ABB RobotStudio station: PROYECTO_SIM_20221117-140459.rsstn

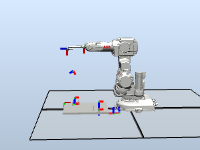
Station PROYECTO_SIM (saved by RobotStudio 6.5.7558.2005)
Controller IRB_140_6kg_0.81m
  mechanical unit ROB_1: IRB140_6_81_C_03, 6 joints, base frame (0, 0, 0) mm
Layout (positions relative to the parent item):
  - IRB140_6_81_C_03 [mechanism, from Robots\IRB140_6_81_C_G_03.rslib] at (0, 0, 0) mm; joint values [0, 0, 0, 0, 0, 0] (rad or m)
  - Herramienta_Proyecto [mechanism, from Libraries\Herramienta_Proyecto.rslib] at (515, 0, 712) mm, rotated rx 0 ry 90 rz 0 deg
  - Placa [part] at (500, 0, 0) mm
Attachment: Herramienta_Proyecto is attached to IRB140_6_81_C_03 / Link6
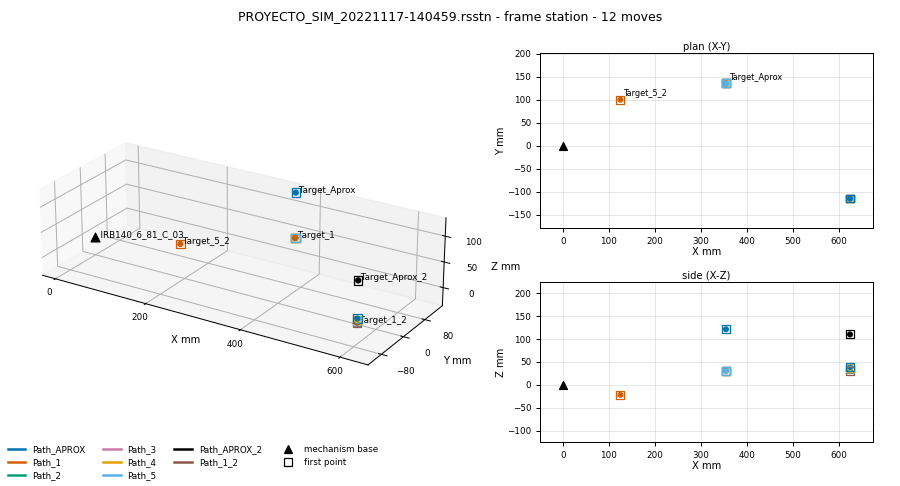
[picture p0: tool path of PROYECTO_SIM_20221117-140459.rsstn in frame station, 12 of 14 moves have a stored position in this frame; points joined in program order, loops and branches not executed]
Targets, tools, work objects and paths stored in the station, written as RAPID:
! task T_ROB1
MODULE CalibData
  PERS tooldata Herramienta_Proyecto_TCP:=[TRUE,[[20,0,187.132],[1,0,0,0]],[0.4,[8.3,90.3,0.6],[1,0,0,0],0,0,0]];
  TASK PERS wobjdata Workobject_1:=[FALSE,TRUE,"",[[750,-215,20],[0,0,1,0]],[[0,0,0],[1,0,0,0]]];
ENDMODULE

! task T_ROB1
MODULE Module1
  CONST jointtarget HOME:=[[0,0,0,0,0,0],[9E+09,9E+09,9E+09,9E+09,9E+09,9E+09]];
  CONST jointtarget MID:=[[0,30,0,0,0,0],[9E+09,9E+09,9E+09,9E+09,9E+09,9E+09]];
  CONST robtarget Target_10:=[[200,200,0],[1,0,0,0],[0,0,0,0],[9E+09,9E+09,9E+09,9E+09,9E+09,9E+09]];
  CONST robtarget Target_Aprox:=[[395.042933274,350.43399652,-101.200003603],[1,0.000000002,0.000000007,-0.000000013],[0,0,0,0],[9E+09,9E+09,9E+09,9E+09,9E+09,9E+09]];
  CONST robtarget Target_2:=[[395.042934534,350.43399616,-11.200003603],[1,0.000000002,0.000000007,-0.000000013],[0,0,0,0],[9E+09,9E+09,9E+09,9E+09,9E+09,9E+09]];
  CONST robtarget Target_1:=[[395.042934534,350.43399616,-11.200003603],[1,0.000000002,0.000000007,-0.000000013],[0,0,0,0],[9E+09,9E+09,9E+09,9E+09,9E+09,9E+09]];
  CONST robtarget Target_3:=[[395.042934534,350.43399616,-11.200003603],[1,0.000000002,0.000000007,-0.000000013],[0,0,0,0],[9E+09,9E+09,9E+09,9E+09,9E+09,9E+09]];
  CONST robtarget Target_4:=[[395.042934534,350.43399616,-11.200003603],[1,0.000000002,0.000000007,-0.000000013],[0,0,0,0],[9E+09,9E+09,9E+09,9E+09,9E+09,9E+09]];
  CONST robtarget Target_5:=[[395.042934534,350.43399616,-11.200003603],[1,0.000000002,0.000000007,-0.000000013],[0,0,0,0],[9E+09,9E+09,9E+09,9E+09,9E+09,9E+09]];
  CONST robtarget Target_Aprox_2:=[[125,100,-90],[1,0,0,0],[0,0,0,0],[9E+09,9E+09,9E+09,9E+09,9E+09,9E+09]];
  CONST robtarget Target_1_2:=[[125,100,-11.15],[1,0,0,0],[0,0,0,0],[9E+09,9E+09,9E+09,9E+09,9E+09,9E+09]];
  CONST robtarget Target_2_2:=[[125,100,-13.62],[1,0,0,0],[0,0,0,0],[9E+09,9E+09,9E+09,9E+09,9E+09,9E+09]];
  CONST robtarget Target_3_2:=[[125,100,-16.45],[1,0,0,0],[0,0,0,0],[9E+09,9E+09,9E+09,9E+09,9E+09,9E+09]];
  CONST robtarget Target_4_2:=[[125,100,-19.15],[1,0,0,0],[0,0,0,0],[9E+09,9E+09,9E+09,9E+09,9E+09,9E+09]];
  CONST robtarget Target_5_2:=[[625,315,41.65],[0,0,1,0],[0,0,0,0],[9E+09,9E+09,9E+09,9E+09,9E+09,9E+09]];
  PROC Path_HOME()
    MoveAbsJ HOME,v1000,z100,Herramienta_Proyecto_TCP\WObj:=wobj0;
  ENDPROC
  PROC Path_MID()
    MoveAbsJ MID,v1000,z100,Herramienta_Proyecto_TCP\WObj:=wobj0;
  ENDPROC
  PROC Path_APROX()
    MoveJ Target_Aprox,v1000,z100,Herramienta_Proyecto_TCP\WObj:=Workobject_1;
  ENDPROC
  PROC Path_1()
    MoveJ Target_1,v1000,z100,Herramienta_Proyecto_TCP\WObj:=Workobject_1;
  ENDPROC
  PROC Path_2()
    MoveJ Target_2,v1000,z100,Herramienta_Proyecto_TCP\WObj:=Workobject_1;
  ENDPROC
  PROC Path_3()
    MoveJ Target_3,v1000,z100,Herramienta_Proyecto_TCP\WObj:=Workobject_1;
  ENDPROC
  PROC Path_4()
    MoveJ Target_4,v1000,z100,Herramienta_Proyecto_TCP\WObj:=Workobject_1;
  ENDPROC
  PROC Path_5()
    MoveJ Target_5,v1000,z100,Herramienta_Proyecto_TCP\WObj:=Workobject_1;
  ENDPROC
  PROC Path_APROX_2()
    MoveJ Target_Aprox_2,v1000,z100,Herramienta_Proyecto_TCP\WObj:=Workobject_1;
  ENDPROC
  PROC Path_1_2()
    MoveJ Target_1_2,v1000,z100,Herramienta_Proyecto_TCP\WObj:=Workobject_1;
  ENDPROC
  PROC Path_2_2()
    MoveJ Target_2_2,v1000,z100,Herramienta_Proyecto_TCP\WObj:=Workobject_1;
  ENDPROC
  PROC Path_3_2()
    MoveJ Target_3_2,v1000,z100,Herramienta_Proyecto_TCP\WObj:=Workobject_1;
  ENDPROC
  PROC Path_4_2()
    MoveJ Target_4_2,v1000,z100,Herramienta_Proyecto_TCP\WObj:=Workobject_1;
  ENDPROC
  PROC Path_5_2()
    MoveJ Target_5_2,v1000,z100,Herramienta_Proyecto_TCP\WObj:=Workobject_1;
  ENDPROC
ENDMODULE

